TYPE "PosFbk_AnalogIn_Alr"
VERSION : 0.1
// Block: PosFbk_AnalogIn_Alr
   STRUCT
      CommFault : Bool;
      SensorFault : Bool;
      Resolution : Bool;
   END_STRUCT;

END_TYPE
